(* PLC project safeApp1, BrAutomation SafeDESIGNER  5.16.0.0 *)
(* stored: companyURL http://www.br-automation.com, creationDateTime Tue Mar 01 14:49:36 2022 *)

PROGRAM Main

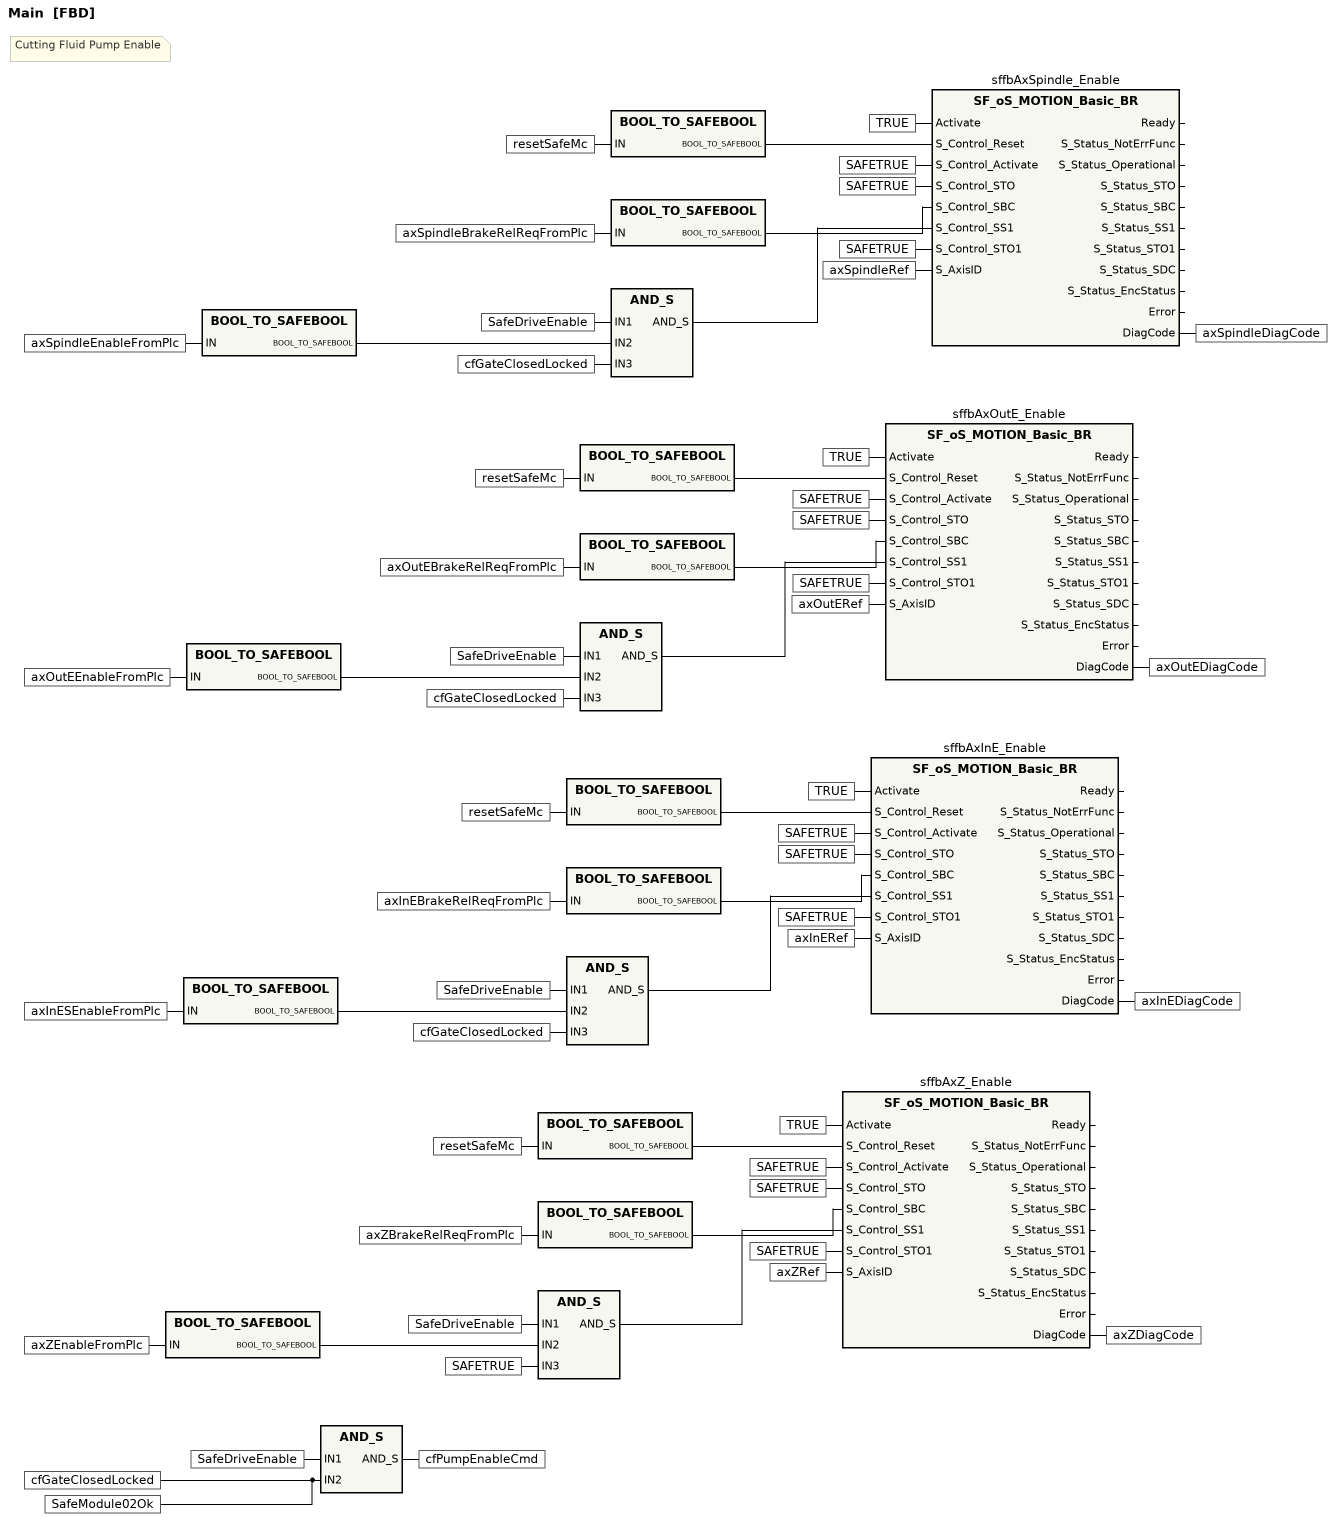
(* FBD diagram, written out as Structured Text *)
sffbAxSpindle_Enable(Activate := TRUE, S_Control_Reset := BOOL_TO_SAFEBOOL(resetSafeMc), S_Control_Activate := SAFETRUE, S_Control_STO := SAFETRUE, S_Control_SBC := BOOL_TO_SAFEBOOL(axSpindleBrakeRelReqFromPlc), S_Control_SS1 := AND_S(SafeDriveEnable, BOOL_TO_SAFEBOOL(axSpindleEnableFromPlc), cfGateClosedLocked), S_Control_STO1 := SAFETRUE, S_AxisID := axSpindleRef);
axSpindleDiagCode := sffbAxSpindle_Enable.DiagCode;
sffbAxOutE_Enable(Activate := TRUE, S_Control_Reset := BOOL_TO_SAFEBOOL(resetSafeMc), S_Control_Activate := SAFETRUE, S_Control_STO := SAFETRUE, S_Control_SBC := BOOL_TO_SAFEBOOL(axOutEBrakeRelReqFromPlc), S_Control_SS1 := AND_S(SafeDriveEnable, BOOL_TO_SAFEBOOL(axOutEEnableFromPlc), cfGateClosedLocked), S_Control_STO1 := SAFETRUE, S_AxisID := axOutERef);
axOutEDiagCode := sffbAxOutE_Enable.DiagCode;
sffbAxInE_Enable(Activate := TRUE, S_Control_Reset := BOOL_TO_SAFEBOOL(resetSafeMc), S_Control_Activate := SAFETRUE, S_Control_STO := SAFETRUE, S_Control_SBC := BOOL_TO_SAFEBOOL(axInEBrakeRelReqFromPlc), S_Control_SS1 := AND_S(SafeDriveEnable, BOOL_TO_SAFEBOOL(axInESEnableFromPlc), cfGateClosedLocked), S_Control_STO1 := SAFETRUE, S_AxisID := axInERef);
axInEDiagCode := sffbAxInE_Enable.DiagCode;
sffbAxZ_Enable(Activate := TRUE, S_Control_Reset := BOOL_TO_SAFEBOOL(resetSafeMc), S_Control_Activate := SAFETRUE, S_Control_STO := SAFETRUE, S_Control_SBC := BOOL_TO_SAFEBOOL(axZBrakeRelReqFromPlc), S_Control_SS1 := AND_S(SafeDriveEnable, BOOL_TO_SAFEBOOL(axZEnableFromPlc), SAFETRUE), S_Control_STO1 := SAFETRUE, S_AxisID := axZRef);
axZDiagCode := sffbAxZ_Enable.DiagCode;
(* Cutting Fluid Pump Enable *)
cfPumpEnableCmd := AND_S(SafeDriveEnable, cfGateClosedLocked, SafeModule02Ok);
END_PROGRAM
